TYPE ST_VelocityBoundary :
STRUCT
	qMin_t : LREAL;
	qMax_t : LREAL;
END_STRUCT
END_TYPE

(* stored: Version 1.1.0.1, ProductVersion 3.1.4022.18
   DUT ST_VelocityBoundary: Id {9d500dd6-66a5-47d9-9bec-f111d3b91175} *)
